FUNCTION MaxOfTwo : INT
VAR_INPUT
	x:INT;
	y:INT;
END_VAR
VAR
END_VAR

IF x>y THEN
	MaxOfTwo := x;
ELSE
	MaxOfTwo := y;
END_IF

END_FUNCTION

(* stored: Version 1.1.0.1, ProductVersion 3.1.4024.16
   POU MaxOfTwo: Id {63d5f10b-dee2-45f9-80f2-faab495396c0}, SpecialFunc None *)
